# EPICS substitutions: apps/mmfeuApp/Db/mmfeusums.substitutions
file "db/mmfeusums.db" {
pattern { SUFFIX }
{ Current_A }
{ XTmpV6 }
{ MTmpInt }
{ TmpSdX }
{ TmpSdA }
}
